{attribute 'GeneratedUsingTerminal: EM7004-0000-0017'}
{attribute addProperty BoxType "EM7004-0000-0017"}
{attribute addProperty Id "EtcSlaveTerminalBaseDI_InputsAT %I*DI_Inputs_9882B61816ENC_Inputs_Channel_1AT %I*ENC_Inputs_Channel_E5B5E92911ENC_Inputs_Channel_2AT %I*ENC_Inputs_Channel_E5B5E92911ENC_Inputs_Channel_3AT %I*ENC_Inputs_Channel_E5B5E92911ENC_Inputs_Channel_4AT %I*ENC_Inputs_Channel_E5B5E92911PLS_InputsAT %I*PLS_Inputs_65C9A3D62DO_OutputsAT %Q*DO_Outputs_47E26D6A16AO_Outputs_Channel_1AT %Q*AO_Outputs_Channel_BA7EBB7C2AO_Outputs_Channel_2AT %Q*AO_Outputs_Channel_BA7EBB7C2AO_Outputs_Channel_3AT %Q*AO_Outputs_Channel_BA7EBB7C2AO_Outputs_Channel_4AT %Q*AO_Outputs_Channel_BA7EBB7C2ENC_Outputs_Channel_1AT %Q*ENC_Outputs_Channel_2E82BC435ENC_Outputs_Channel_2AT %Q*ENC_Outputs_Channel_2E82BC435ENC_Outputs_Channel_3AT %Q*ENC_Outputs_Channel_2E82BC435ENC_Outputs_Channel_4AT %Q*ENC_Outputs_Channel_2E82BC435PLS_OutputsAT %Q*PLS_Outputs_8EABC2241WcStateAT %I*WcState_9091E0EB2InfoDataAT %I*InfoData_32EB74EA10"}
{attribute addProperty CRC "1336621591"}
{attribute addProperty Size "119"}
TYPE EM7004_4FAB3A17 EXTENDS EtcSlaveTerminalBase :
STRUCT
	{attribute addProperty Name "DI_Inputs"}
	DI_Inputs : DI_Inputs_9882B618;
	{attribute addProperty Name "ENC_Inputs_Channel_1"}
	ENC_Inputs_Channel_1 : ENC_Inputs_Channel_E5B5E929;
	{attribute addProperty Name "ENC_Inputs_Channel_2"}
	ENC_Inputs_Channel_2 : ENC_Inputs_Channel_E5B5E929;
	{attribute addProperty Name "ENC_Inputs_Channel_3"}
	ENC_Inputs_Channel_3 : ENC_Inputs_Channel_E5B5E929;
	{attribute addProperty Name "ENC_Inputs_Channel_4"}
	ENC_Inputs_Channel_4 : ENC_Inputs_Channel_E5B5E929;
	{attribute addProperty Name "PLS_Inputs"}
	PLS_Inputs : PLS_Inputs_65C9A3D6;
	{attribute addProperty Name "DO_Outputs"}
	DO_Outputs : DO_Outputs_47E26D6A;
	{attribute addProperty Name "AO_Outputs_Channel_1"}
	AO_Outputs_Channel_1 : AO_Outputs_Channel_BA7EBB7C;
	{attribute addProperty Name "AO_Outputs_Channel_2"}
	AO_Outputs_Channel_2 : AO_Outputs_Channel_BA7EBB7C;
	{attribute addProperty Name "AO_Outputs_Channel_3"}
	AO_Outputs_Channel_3 : AO_Outputs_Channel_BA7EBB7C;
	{attribute addProperty Name "AO_Outputs_Channel_4"}
	AO_Outputs_Channel_4 : AO_Outputs_Channel_BA7EBB7C;
	{attribute addProperty Name "ENC_Outputs_Channel_1"}
	ENC_Outputs_Channel_1 : ENC_Outputs_Channel_2E82BC43;
	{attribute addProperty Name "ENC_Outputs_Channel_2"}
	ENC_Outputs_Channel_2 : ENC_Outputs_Channel_2E82BC43;
	{attribute addProperty Name "ENC_Outputs_Channel_3"}
	ENC_Outputs_Channel_3 : ENC_Outputs_Channel_2E82BC43;
	{attribute addProperty Name "ENC_Outputs_Channel_4"}
	ENC_Outputs_Channel_4 : ENC_Outputs_Channel_2E82BC43;
	{attribute addProperty Name "PLS_Outputs"}
	PLS_Outputs : PLS_Outputs_8EABC224;
	{attribute addProperty Name "WcState"}
	WcState : WcState_9091E0EB;
	{attribute addProperty Name "InfoData"}
	InfoData : InfoData_32EB74EA;
END_STRUCT
END_TYPE

(* stored: Version 1.2.0.0, ProductVersion 3.1.4024.9
   DUT EM7004_4FAB3A17: Id {14b2655a-b3ad-432a-9ec4-42d55f6e1355} *)
